TYPE ST_CAMERA_Evaluation :
STRUCT
	nTotalReads			: UDINT;
	nReadCodes			: UDINT;
	nNOKCodes			: UDINT;

	nGoodCodes			: UDINT;
	nFairCodes			: UDINT;
	nPoorCodes			: UDINT;

	fReadEfficiency			: LREAL;
	fNOKEfficiency			: LREAL;

	fGoodEfficiency		: LREAL;
	fFairEfficiency			: LREAL;
	fPoorEfficiency			: LREAL;

END_STRUCT
END_TYPE

(* stored: Version 1.1.0.1
   DUT ST_CAMERA_Evaluation: Id {c0d4c0cd-c971-4164-8201-8f16624f9f28} *)
